// TwinCAT 3 PLC project MainPLC
// ProgramVersion: 3.1.4024.12
// libraries:
//   Tc2_Standard, * (Beckhoff Automation GmbH)
//   Tc2_System, * (Beckhoff Automation GmbH)
//   Tc2_Utilities, * (Beckhoff Automation GmbH)
//   Tc3_Module, * (Beckhoff Automation GmbH)
// project tree:
//   DUTs/ User1DUT.TcDUT, User2DUT.TcDUT, UserInnerInnerDUT.TcDUT, UserInnerInnerDUTPersistent.TcDUT
//   GVLs/ GVL.TcGVL
//   / PlcTask.TcTTO
//   POUs/ MAIN.TcPOU, TestFB1.TcPOU, TestFB1Device.TcPOU, TestFB1DeviceSubdevice.TcPOU
// real-time tasks:
//   TASK PlcTask: cycle T#10ms, priority 20, ADS port 350

CONFIGURATION MainPLC
    RESOURCE PLC ON TwinCAT3
        TASK PlcTask(INTERVAL := T#10ms, PRIORITY := 20);
        PROGRAM MAIN WITH PlcTask : MAIN;
    END_RESOURCE
END_CONFIGURATION

// ---- DUTs/User1DUT.TcDUT
TYPE User1DUT :
STRUCT
	Int1:INT:=157;
	Int2:INT:=168;
	Bool1:BOOL:=TRUE;
	InInVar:UserInnerInnerDUT;
	Bool2:BOOL:=TRUE;
	Bool3:BOOL:=FALSE;
END_STRUCT
END_TYPE

// ---- DUTs/User2DUT.TcDUT
TYPE User2DUT :
STRUCT
	Int1:INT:=157;
	Int2:INT:=168;
	Bool1:BOOL:=TRUE;
	InInVar:UserInnerInnerDUTPersistent;
	Bool2:BOOL:=TRUE;
	Bool3:BOOL:=FALSE;
END_STRUCT
END_TYPE

// ---- DUTs/UserInnerInnerDUT.TcDUT
TYPE UserInnerInnerDUT :
STRUCT
	IntInIn1:INT:=12;
	RealInIn1:REAL:=123.2345;	
END_STRUCT
END_TYPE

// ---- DUTs/UserInnerInnerDUTPersistent.TcDUT
TYPE UserInnerInnerDUTPersistent :
STRUCT PERSISTENT
	IntInIn1_Pers:INT:=321;
	RealInIn1_Pers:REAL:=321.9;	
END_STRUCT
END_TYPE

// ---- GVLs/GVL.TcGVL
{attribute 'qualified_only'}
VAR_GLOBAL PERSISTENT
	PersVarGlobalArray: ARRAY [0..3] OF INT := [6,7,8];  //Global variable, Persistent, Array 0..3 of INT
	PersVarGlobalBool1:BOOL:=TRUE;  //Global variable, Persistent, BOOL
	PersVarGlobalBool2:BOOL:=FALSE; //Global variable, Persistent, BOOL
	PersVarGlobalTime1:TIME:=T#300MS; //Global variable, Persistent, TIME
	PersVarGlobalUser1_1:User1DUT; //Global variable, Top element Persistent, User data type "User1DUT", 2 level nested structure, Non of the children defined explicitly as persistent, but should inherit Persistent status from Top Element/Parent
	DatetimeUTC : DT;
	Datetime : DT;
	ActualDate : DATE;
	ActualTime : TIME;
	ActualLTime : LTIME;
END_VAR

VAR_GLOBAL
	NonPersVarGlobalBool3:BOOL:=TRUE;  //Global variable Non Persistent BOOL
	NonPersVarGlobalBool4:BOOL:=FALSE; //Global variable Non Persistent BOOL
	NonPersVarGlobalUser1_2:User1DUT; //Global variable, Top element Non Persistent, User data type "User1DUT", 2 level nested structure, None of the children defined explicitly as persistent
	MixedPersVarGlobalUser1_3:User2DUT;  //User defined data type, Top element Non Persistent, User data type "User2DUT", 2 level nested structure, Some children devined as persistent - mixed status 
END_VAR

// ---- POUs/MAIN.TcPOU
PROGRAM MAIN
VAR
	NonPersMainVarBool1:BOOL:=TRUE;
	NonPersMainVarBool2:BOOL:=FALSE;
	TestFB1_DB1:TestFB1;
	
	fbToLocal 		: FB_FileTimeToTzSpecificLocalTime;
	fileTime        : T_FILETIME;
	fbGetSystemTime : GETSYSTEMTIME;
END_VAR
VAR PERSISTENT
	PersMainVarBool3:BOOL:=TRUE;
	PersMainVarBool4:BOOL:=FALSE;
	PersMainVarInt1:INT:=0;
END_VAR


PersMainVarInt1:=PersMainVarInt1+1;
TestFB1_DB1(I_Run:=TRUE);

fbGetSystemTime(timeLoDW=>fileTime.dwLowDateTime, timeHiDW=>fileTime.dwHighDateTime );
GVL.DatetimeUTC := FILETIME_TO_DT(fileTime);
fbToLocal( in := fileTime, tzInfo := WEST_EUROPE_TZI );
GVL.Datetime := FILETIME_TO_DT( fbToLocal.out );
GVL.ActualDate := DT_TO_DATE(GVL.Datetime);
GVL.ActualTime := DT_TO_TIME(GVL.Datetime);
GVL.ActualLTime := TIME_TO_LTIME(GVL.ActualTime);

END_PROGRAM

// ---- POUs/TestFB1.TcPOU
FUNCTION_BLOCK TestFB1
VAR_INPUT
	I_Run:BOOL;
END_VAR
VAR_OUTPUT PERSISTENT
	O_Number:INT;
END_VAR
VAR
	Inst_TestFB1Device:TestFB1Device;
	FB_Internal:INT;
	FB_InternalStatic:INT:=123;
END_VAR
VAR PERSISTENT
	BP_tSetup:TIME:=T#300MS;
	BP_iSetup:INT:=67;
END_VAR

IF I_Run THEN
	O_Number:=O_Number +1;
	FB_Internal:=Fb_Internal+3;
END_IF
Inst_TestFB1Device();

END_FUNCTION_BLOCK

// ---- POUs/TestFB1Device.TcPOU
FUNCTION_BLOCK TestFB1Device
VAR_INPUT
END_VAR
VAR_OUTPUT
END_VAR
VAR
	Inst_Subdevice1:TestFB1DeviceSubdevice;
	NonPerstInt1:INT:=9;
	NonPerstInt2:INT:=10;
END_VAR
VAR PERSISTENT
	PersInt1:INT:=435;
END_VAR

NonPerstInt1:=NonPerstInt1+1;
Inst_Subdevice1();

END_FUNCTION_BLOCK

// ---- POUs/TestFB1DeviceSubdevice.TcPOU
FUNCTION_BLOCK TestFB1DeviceSubdevice
VAR_INPUT
END_VAR
VAR_OUTPUT
END_VAR
VAR
	NonPerstInt1:INT:=9;
	NonPerstInt2:INT:=10;
END_VAR
VAR PERSISTENT
	PersInt1:INT:=435;
END_VAR

PersInt1:=PersInt1+1;

END_FUNCTION_BLOCK
